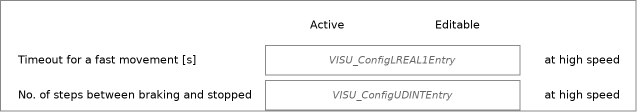
VISUALIZATION VISU_M2Config_ZAxis_Specific  // 637x112
VAR_IN_OUT
    editable : M2ZAxisConfig;
	active : M2ZAxisConfig;
END_VAR
    Frame (265,80 255x30), tooltip "The number of steps to be expected between the time at which the PLC realizes that the brake signal must be set, and the time that the axis is fully stopped (for Z axis: at low speed)"
        shows VISU_ConfigUDINTEntry(active := active.highSpeedStoppingSteps, editable := editable.highSpeedStoppingSteps)
    Label (15,80 250x30), "No. of steps between braking and stopped"
    Label (530,80 105x30), "at high speed"
    Frame (265,45 255x30), tooltip "Time (in seconds) to wait after the axis has been moved"
        shows VISU_ConfigLREAL1Entry(active := active.highSpeedTimeout, editable := editable.highSpeedTimeout)
    Label (15,45 285x30), "Timeout for a fast movement [s]"
    Label (530,45 105x30), "at high speed"
    Label (265,15 125x20), "Active"
    Label (395,15 125x20), "Editable"
END_VISUALIZATION

(* stored: Version 1.1.0.1, ProductVersion 3.1.4019.2
   Visu VISU_M2Config_ZAxis_Specific: Id {1df49191-ce99-4857-b3c2-efdaf3baf2b4} *)
